FUNCTION_BLOCK Kulbana_composit
  (* Version 1.0, 2005-07-13, Goran Cengic, Chalmers *)
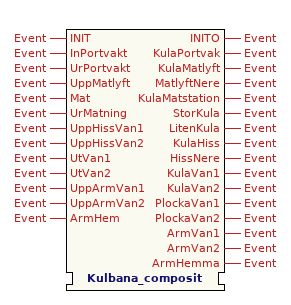
  EVENT_INPUT
    INIT;
    InPortvakt;
    UrPortvakt;
    UppMatlyft;
    Mat;
    UrMatning;
    UppHissVan1;
    UppHissVan2;
    UtVan1;
    UtVan2;
    UppArmVan1;
    UppArmVan2;
    ArmHem;
  END_EVENT
  EVENT_OUTPUT
    INITO;
    KulaPortvak;
    KulaMatlyft;
    MatlyftNere;
    KulaMatstation;
    StorKula;
    LitenKula;
    KulaHiss;
    HissNere;
    KulaVan1;
    KulaVan2;
    PlockaVan1;
    PlockaVan2;
    ArmVan1;
    ArmVan2;
    ArmHemma;
  END_EVENT
  FBS
    cycle : E_CYCLE;
    initsplit : E_SPLIT2;
    adlink : ADLINK_IO;
    split7 : E_SPLIT7;
    merge7 : E_MERGE7;
    pv : PV_model;
    ml : ML_model;
    ms : MS_model;
    hs : HS_model;
    vn1 : VN_model;
    vn2 : VN_model;
    ar : AR_model;
  END_FBS
  EVENT_CONNECTIONS
    INIT TO initsplit.EI;
    initsplit.EO1 TO INITO;
    initsplit.EO2 TO cycle.START;
    cycle.EO TO adlink.READ;
    adlink.VALUES TO split7.EI;
    split7.EO1 TO pv.Values;
    split7.EO2 TO ml.Values;
    split7.EO3 TO ms.Values;
    split7.EO4 TO hs.Values;
    split7.EO5 TO vn1.Values;
    split7.EO6 TO vn2.Values;
    split7.EO7 TO ar.Values;
    pv.Write TO merge7.EI1;
    ml.Write TO merge7.EI2;
    ms.Write TO merge7.EI3;
    hs.Write TO merge7.EI4;
    vn1.Write TO merge7.EI5;
    vn2.Write TO merge7.EI6;
    ar.Write TO merge7.EI7;
    merge7.EO TO adlink.WRITE;
    InPortvakt TO pv.InPortvakt;
    UrPortvakt TO pv.UrPortvakt;
    pv.KulaPortvakt TO KulaPortvakt;
    UppMatlyft TO ml.UppMatlyft;
    ml.KulaMatlyft TO KulaMatlyft;
    ml.MatlyftNere TO MatlyftNere;
    Mat TO ms.Mat;
    UrMatning TO ms.UrMatning;
    ms.KulaMatstation TO KulaMatstation;
    ms.StorKula TO StorKula;
    ms.LitenKula TO LitenKula;
    UppHissVan1 TO hs.UppHissVan1;
    UppHissVan2 TO hs.UppHissVan2;
    hs.KulaHiss TO KulaHiss;
    hs.KulaVan1 TO KulaVan1;
    hs.KulaVan2 TO KulaVan2;
    hs.HissNere TO HissNere;
    UtVan1 TO vn1.UtVan;
    vn1.PlockaVan TO PlockaVan1;
    UtVan2 TO vn2.UtVan;
    vn2.PlockaVan TO PlockaVan2;
    UppArmVan1 TO ar.UppArmVan1;
    UppArmVan2 TO ar.UppArmVan2;
    ArmHem TO ar.ArmHem;
    ar.ArmVan1 TO ArmVan1;
    ar.ArmVan2 TO ArmVan2;
    ar.ArmHemma TO ArmHemma;
  END_CONNECTIONS
  DATA_CONNECTIONS
    200 TO cycle.DT;
    adlink.INPUT0 TO pv.KulaPortvakt_sig;
    pv.InPortvakt_sig TO adlink.OUTPUT0;
    pv.UrPortvakt_sig TO adlink.OUTPUT1;
    adlink.INPUT1 TO ml.MatlyftNere_sig;
    adlink.INPUT2 TO ml.KulaMatlyft_sig;
    adlink.INPUT3 TO ml.MatlyftUppe_sig;
    adlink.INPUT4 TO ml.KulaMatstation_sig;
    ml.UppMatlyft_sig TO adlink.OUTPUT2;
    adlink.INPUT4 TO ms.KulaMatstation_sig;
    adlink.INPUT5 TO ms.StorKula_sig;
    adlink.INPUT6 TO ms.LitenKula_sig;
    ms.Mat_sig TO adlink.OUTPUT4;
    ms.UrMatning_sig TO adlink.OUTPUT3;
    adlink.INPUT7 TO hs.HissNere_sig;
    adlink.INPUT10 TO hs.KulaHiss_sig;
    adlink.INPUT11 TO hs.HissVan1_sig;
    adlink.INPUT12 TO hs.KulaVan1_sig;
    adlink.INPUT14 TO hs.HissVan2_sig;
    adlink.INPUT15 TO hs.KulaVan2_sig;
    hs.UppHissVan1_sig TO adlink.OUTPUT5;
    hs.UppHissVan2_sig TO adlink.OUTPUT6;
    adlink.INPUT12 TO vn1.KulaVan_sig;
    adlink.INPUT13 TO vn1.PlockaVan_sig;
    adlink.INPUT22 TO vn1.KulaFast_sig;
    adlink.INPUT20 TO vn1.ArmVan_sig;
    adlink.INPUT17 TO vn1.ArmHemma_sig;
    vn1.UtVan_sig TO adlink.OUTPUT7;
    vn1.LyftVan_sig TO adlink.OUTPUT10;
    adlink.INPUT15 TO vn2.KulaVan_sig;
    adlink.INPUT16 TO vn2.PlockaVan_sig;
    adlink.INPUT22 TO vn2.KulaFast_sig;
    adlink.INPUT21 TO vn2.ArmVan_sig;
    adlink.INPUT17 TO vn2.ArmHemma_sig;
    vn2.UtVan_sig TO adlink.OUTPUT11;
    vn2.LyftVan_sig TO adlink.OUTPUT12;
    adlink.INPUT20 TO ar.ArmVan1_sig;
    adlink.INPUT13 TO ar.KulaVan1_sig;
    adlink.INPUT21 TO ar.ArmVan2_sig;
    adlink.INPUT16 TO ar.KulaVan2_sig;
    adlink.INPUT22 TO ar.KulaFast_sig;
    adlink.INPUT17 TO ar.ArmHemma_sig;
    ar.UppArmVan1_sig TO adlink.OUTPUT13;
    ar.UppArmVan2_sig TO adlink.OUTPUT14;
    ar.VridArmHoger_sig TO adlink.OUTPUT15;
    ar.Sug_sig TO adlink.OUTPUT16;
  END_CONNECTIONS
END_FUNCTION_BLOCK
(* other elements stored in the file *)
(* Values split *)
(* Write merge *)
(* Portvakt *)
(* Matlyft *)
(* Matstation *)
(* Hiss *)
(* Vaning 1 *)
(* Vaning 2 *)
(* Arm *)
(* Portvakt signals *)
(* Matlyft signals *)
(* Matstation signals *)
(* Hiss signal *)
(* Vaning 1 signals *)
(* Vaning 2 signals *)
(* Arm signals *)
